(* IEC 61131-3 sources: ATCMcontrol_Engineering/src/TargetBase/Libs/ATCM_IEC1131_3/table_24, 7 files *)

(* ---- add.st ---- *)
(*[[
    UserURL= "ATCMfile:ADD.htm"
]]*)

FUNCTION ADD : ANY_MAGNITUDE
VAR_INPUT
    IN1 : ANY_MAGNITUDE;
END_VAR
VAR_IN_EXT
    IN2 : ANY_MAGNITUDE;
END_VAR

inline +

END_FUNCTION

(* ---- div.st ---- *)
(*[[
    UserURL= "ATCMfile:DIV.htm"
]]*)

FUNCTION DIV : ANY_NUM
VAR_INPUT
    IN1: ANY_NUM;
    IN2: ANY_NUM;
END_VAR

inline /

END_FUNCTION

(* ---- expt.st ---- *)
(*[[
    UserURL= "ATCMfile:EXPT.htm"
]]*)

FUNCTION EXPT : ANY_REAL
VAR_INPUT
    IN1: ANY_REAL;
    IN2: ANY_NUM;
END_VAR

overload REAL(REAL,DINT)    inline
{
    %1
    %2
    pow_real_dint
}
overload REAL(REAL,INT)     inline
{
    %1
    %2
    pow_real_int
}
overload LREAL(LREAL,DINT)  inline
{
    %1
    %2
    pow_lreal_dint
}
overload LREAL(LREAL,INT)   inline
{
    %1
    %2
    pow_lreal_int
}
overload REAL(REAL,REAL)    inline
{
    %1
    %2
    pow_real_real
}
overload LREAL(LREAL,LREAL) inline
{
    %1
    %2
    pow_lreal_lreal
}
overload REAL(REAL,LREAL)   inline
{
    %1
    real_to_lreal
    %2
    pow_lreal_lreal
    lreal_to_real
}
overload LREAL(LREAL,REAL)  inline
{
    %1
    %2
    real_to_lreal
    pow_lreal_lreal
}

END_FUNCTION

(* ---- mod.st ---- *)
(*[[
    UserURL= "ATCMfile:MOD.htm"
]]*)

FUNCTION MOD : ANY_INT
VAR_INPUT
    IN1: ANY_INT;
    IN2: ANY_INT;
END_VAR

inline MOD

END_FUNCTION

(* ---- move.st ---- *)
FUNCTION MOVE: ANY
VAR_INPUT
    In: ANY;
END_VAR

inline :=

END_FUNCTION

(* ---- mul.st ---- *)
(*[[
    UserURL= "ATCMfile:MUL.htm"
]]*)

FUNCTION MUL : ANY_NUM
VAR_INPUT
    IN1 : ANY_NUM;
END_VAR
VAR_IN_EXT
    IN2 : ANY_NUM;
END_VAR

inline *

END_FUNCTION

(* ---- sub.st ---- *)
(*[[
    UserURL= "ATCMfile:SUB.htm"
]]*)

FUNCTION SUB : ANY_MAGNITUDE
VAR_INPUT
    IN1: ANY_MAGNITUDE;
    IN2: ANY_MAGNITUDE;
END_VAR

inline -

END_FUNCTION
